Yaskawa INFORM job: OK_R2_O7,1(180,-90)OKKR_COMOUT.JBI

/JOB
//NAME OK_R2_O7,1(180,-90)OKKR_COMOUT
///FOLDERNAME X4
//POS
///NPOS 62,62,62,4,0,0
///TOOL 0
///POSTYPE PULSE
///PULSE
C00000=-125435,-77622,-99768,3556,84592,-1364
C00001=-127461,5107,-41648,6005,105402,-2311
C00002=-127602,-5081,-33811,5791,95110,-2850
C00003=-127461,-1910,-29167,5755,93871,-2860
C00004=-127461,-2146,-28156,5750,93132,-2895
C00005=-127461,-2037,-28638,5753,93482,-2879
C00006=-127360,629,-26422,5741,93484,-2844
C00007=-127461,-2008,-28767,5752,93576,-2874
C00008=-103998,1569,-25784,1957,92494,4742
C00009=-103998,1725,-26420,1958,92965,4749
C00010=-103998,1431,-25178,1956,92049,4737
C00011=-103998,1527,-25606,1957,92361,4742
C00012=-104229,4022,-23485,1997,92343,4666
C00013=-103998,1569,-25784,1957,92494,4742
C00014=-86679,-5363,-42434,-983,99074,10321
C00015=-62381,-14690,-36345,-9691,68856,-1615
C00016=-59861,14391,-7375,-13691,69257,-1127
C00017=-59861,14324,-5508,-13799,68107,-994
C00018=-59861,14327,-5726,-13788,68239,-1009
C00019=-59003,16580,-3664,-14156,68277,-700
C00020=-59755,14625,-6291,-13788,68745,-1031
C00021=-56899,7873,-12330,-14940,69480,-85
C00022=-55561,14142,-1887,-19350,68569,3889
C00023=-55984,15101,-1014,-19198,68428,3753
C00024=-55363,11408,-6012,-19288,69688,3774
C00025=-80499,-60483,-73568,-30648,97810,39569
C00026=-157567,-32017,-43550,-5241,58907,29882
C00027=-159996,-19727,-31763,-3894,57836,28984
C00028=-159996,-19632,-29676,-3947,56602,29029
C00029=-159996,-19645,-29901,-3941,56733,29024
C00030=-161459,-17871,-28596,-3080,56777,28442
C00031=-159996,-19645,-29901,-3941,56733,29024
C00032=-162143,-27333,-35707,-2694,56268,28184
C00033=-172681,-22690,-29875,17242,58260,14469
C00034=-172217,-21488,-29011,16987,58245,14658
C00035=-172321,-29251,-38222,16755,59878,14872
C00036=-170408,-23967,-31499,12392,55434,14706
C00037=-173810,-15316,-27557,19160,62810,14938
C00038=-170769,-6668,-20835,17665,62424,16063
C00039=-175825,-34683,-42059,20272,62319,14051
C00040=-166969,-54255,-34798,10244,21853,14480
C00041=-158903,-38412,-25890,-18291,26979,29827
C00042=-164397,-33556,-23512,2003,33361,24818
C00043=-170768,-56544,-33416,31030,22960,3886
C00044=-164207,-68143,-67141,2531,61479,16355
C00045=-79680,-75357,-72042,-32019,81856,-6685
C00046=-58622,-2742,-23483,-15327,69388,-15208
C00047=-58657,12974,-6767,-15536,67243,-14934
C00048=-62250,22223,1809,-14026,66090,-16116
C00049=-55419,-2669,-22327,-16741,69351,-14036
C00050=-47481,-9553,-15824,-35272,55767,14560
C00051=-66607,-8323,-12437,3279,42530,-8847
C00052=-66424,-8718,-12364,3138,42277,-8766
C00053=-66424,-7242,-5690,3358,38933,-8897
C00054=-61045,-16419,-29917,-8636,63731,-1843
C00055=-128613,-3227,-31039,5936,94424,-3210
C00056=-127935,508,-25861,5822,93118,-3048
C00057=-127978,405,-27754,5840,94227,-3010
C00058=-128179,-4770,-30252,5859,93124,-3128
C00059=-103810,3962,-22936,1928,91967,4796
C00060=-103028,-2446,-34673,1809,95878,5107
C00061=-101377,-7611,-58668,1615,107954,5791
BC00000=203857,716034,897320
BC00001=194529,717607,1053854
BC00002=194529,717607,1053854
BC00003=194529,717607,1053854
BC00004=194529,717607,1053854
BC00005=194529,717607,1053854
BC00006=194529,717607,1053854
BC00007=194529,717607,1053854
BC00008=194529,717607,1053854
BC00009=194529,717607,1053854
BC00010=194529,717607,1053854
BC00011=194529,717607,1053854
BC00012=194529,717607,1053854
BC00013=194529,717607,1053854
BC00014=194529,717607,1053854
BC00015=194529,709946,905441
BC00016=194529,709946,905441
BC00017=194529,709946,905441
BC00018=194529,709946,905441
BC00019=194529,709946,905441
BC00020=194529,709946,905441
BC00021=194529,709946,905441
BC00022=194529,709946,905441
BC00023=194529,709946,905441
BC00024=194529,709946,905441
BC00025=194529,709946,905441
BC00026=194529,709946,905441
BC00027=194529,709946,905441
BC00028=194529,709946,905441
BC00029=194529,709946,905441
BC00030=194529,709946,905441
BC00031=194529,709946,905441
BC00032=194529,709946,905441
BC00033=194529,709946,905441
BC00034=194529,709946,905441
BC00035=194529,709946,905441
BC00036=194529,709946,905441
BC00037=194529,709946,905441
BC00038=194529,709946,905441
BC00039=194529,709946,905441
BC00040=194529,709946,905441
BC00041=194529,709946,905437
BC00042=194529,709946,905437
BC00043=194529,709946,905441
BC00044=194529,709946,905441
BC00045=194529,709946,905441
BC00046=194529,709946,905441
BC00047=194529,709946,905441
BC00048=194529,709946,905441
BC00049=194529,709946,905441
BC00050=194529,709946,905441
BC00051=194529,709946,905441
BC00052=194529,709946,905441
BC00053=194529,709946,905441
BC00054=194529,709946,905441
BC00055=194529,717607,1053854
BC00056=194529,717607,1053854
BC00057=194529,717607,1053854
BC00058=194529,717607,1053854
BC00059=194529,717607,1053854
BC00060=194529,717607,1053854
BC00061=194529,717607,1053854
EC00000=1444023,-556474
EC00001=1319431,-556474
EC00002=1319431,-556474
EC00003=1319431,-556474
EC00004=1319431,-556474
EC00005=1319431,-556474
EC00006=1319431,-556474
EC00007=1319431,-556474
EC00008=1319431,-556474
EC00009=1319431,-556474
EC00010=1319431,-556474
EC00011=1319431,-556474
EC00012=1319431,-556474
EC00013=1319431,-556474
EC00014=1319431,-556474
EC00015=1506869,-556474
EC00016=1506869,-556474
EC00017=1506869,-556474
EC00018=1506869,-556474
EC00019=1506869,-556474
EC00020=1506869,-556474
EC00021=1506869,-556474
EC00022=1506869,-556474
EC00023=1506869,-556474
EC00024=1506869,-556474
EC00025=1506869,-556474
EC00026=1506869,-556474
EC00027=1506869,-556474
EC00028=1506869,-556474
EC00029=1506869,-556474
EC00030=1506869,-556474
EC00031=1506869,-556474
EC00032=1506869,-556474
EC00033=1506869,-556474
EC00034=1506869,-556474
EC00035=1506869,-556474
EC00036=1506869,-556474
EC00037=1506869,-556474
EC00038=1506869,-556474
EC00039=1506869,-556474
EC00040=1506869,-556474
EC00041=1506869,-556474
EC00042=1506869,-556474
EC00043=1506869,-556474
EC00044=1506869,-556474
EC00045=1506869,-556474
EC00046=1506869,-556474
EC00047=1506869,-556474
EC00048=1506869,-556474
EC00049=1506869,-556474
EC00050=1506869,-556474
EC00051=1506869,-556474
EC00052=1506869,-556474
EC00053=1506869,-556474
EC00054=1506869,-556474
EC00055=1319431,-556474
EC00056=1319431,-556474
EC00057=1319431,-556474
EC00058=1319431,-556474
EC00059=1319431,-556474
EC00060=1319431,-556474
EC00061=1319431,-556474
///POSTYPE BASE
///RECTAN
///RCONF 0,0,0,0,0,0,0,0,0,0,0,0,0,0,0,0,0,0,0,0,0,0,0,0
P00006=0.222,-3.123,-1.508,0.0000,0.0000,0.0000
P00021=-0.225,-6.128,-0.405,0.0000,0.0000,0.0000
P00040=-0.030,9.648,2.467,0.0000,0.0000,0.0000
P00041=0.192,3.924,0.305,0.0000,0.0000,0.0000
//INST
///DATE 2024/10/03 09:02
///ATTR SC,RW
///GROUP1 RB1,BS1
///GROUP2 ST1
NOP
'OK_r2_O7.1(180,-90)
'Path S1428
SFTOF3D
MOVJ C00000 BC00000 VJ=100.00  +MOVJ EC00000 VJ=100.00
MOVJ C00001 BC00001 VJ=100.00  +MOVJ EC00001 VJ=100.00
MOVJ C00002 BC00002 VJ=100.00  +MOVJ EC00002 VJ=100.00
SMOVL C00003 BC00003 V=100.0  +MOVJ EC00003
SREFP 3 C00004 BC00004  +REFP EC00004
CALL JOB:SEARCH-R1-S13D
SET P021 P006
SFTON3D P021
SMOVL C00005 BC00005 V=100.0  +MOVJ EC00005
SREFP 3 C00006 BC00006  +REFP EC00006
CALL JOB:SEARCH-R1-S13D
SET P021 P006
SFTON3D P021
SMOVL C00007 BC00007 V=100.0  +MOVJ EC00007
MOVL C00008 BC00008 V=1000.0  +MOVJ EC00008 VJ=100.00
SMOVL C00009 BC00009 V=100.0  +MOVJ EC00009
SREFP 3 C00010 BC00010  +REFP EC00010
CALL JOB:SEARCH-R1-S13D
SET P021 P006
SFTON3D P021
SMOVL C00011 BC00011 V=100.0  +MOVJ EC00011
SREFP 3 C00012 BC00012  +REFP EC00012
CALL JOB:SEARCH-R1-S13D
SET P021 P006
SFTON3D P021
SMOVL C00013 BC00013 V=100.0  +MOVJ EC00013
MOVJ C00014 BC00014 VJ=50.00  +MOVJ EC00014 VJ=50.00
MOVJ C00015 BC00015 VJ=50.00  +MOVJ EC00015 VJ=50.00
SFTOF3D
SMOVL C00016 BC00016 V=166.7  +MOVJ EC00016
SREFP 3 C00017 BC00017  +REFP EC00017
CALL JOB:SEARCH-R1-S13D
SET P040 P006
SFTON3D P040
SMOVL C00018 BC00018 V=100.0  +MOVJ EC00018
SREFP 3 C00019 BC00019  +REFP EC00019
CALL JOB:SEARCH-R1-S13D
SET P040 P006
SFTON3D P040
SMOVL C00020 BC00020 V=100.0  +MOVJ EC00020
SMOVL C00021 BC00021 V=166.7  +MOVJ EC00021
SMOVL C00022 BC00022 V=166.7  +MOVJ EC00022
SREFP 3 C00023 BC00023  +REFP EC00023
CALL JOB:SEARCH-R1-S13D
SET P040 P006
SFTON3D P040
SMOVL C00024 BC00024 V=166.7  +MOVJ EC00024
SFTOF3D
MOVJ C00025 BC00025 VJ=50.00  +MOVJ EC00025 VJ=50.00
MOVJ C00026 BC00026 VJ=50.00  +MOVJ EC00026 VJ=50.00
SMOVL C00027 BC00027 V=166.7  +MOVJ EC00027
SREFP 3 C00028 BC00028  +REFP EC00028
CALL JOB:SEARCH-R1-S13D
SET P041 P006
SFTON3D P041
SMOVL C00029 BC00029 V=100.0  +MOVJ EC00029
SREFP 3 C00030 BC00030  +REFP EC00030
CALL JOB:SEARCH-R1-S13D
SET P040 P041
SFTON3D P041
SMOVL C00031 BC00031 V=100.0  +MOVJ EC00031
SMOVL C00032 BC00032 V=166.7  +MOVJ EC00032
SMOVL C00033 BC00033 V=166.7  +MOVJ EC00033
SREFP 3 C00034 BC00034  +REFP EC00034
CALL JOB:SEARCH-R1-S13D
SET P041 P006
SFTON3D P041
SMOVL C00035 BC00035 V=166.7  +MOVJ EC00035
SFTOF3D
SFTON3D P041
MACRO1 MJ#(0) ARGF14
SMOVL C00036 BC00036 V=166.7  +MOVJ EC00036
ARCON
SMOVL C00037 BC00037 V=8.3  +MOVJ EC00037
SMOVL C00038 BC00038 V=8.3  +MOVJ EC00038
ARCOF
SMOVL C00039 BC00039 V=250.0  +MOVJ EC00039
SMOVL C00040 BC00040 V=250.0  +MOVJ EC00040
SMOVL C00041 BC00041 V=133.3 PL=0  +MOVJ EC00041
ARCON
SMOVL C00042 BC00042 V=9.2  +MOVJ EC00042
ARCOF
SMOVL C00043 BC00043 V=250.0  +MOVJ EC00043
MOVJ C00044 BC00044 VJ=50.00  +MOVJ EC00044 VJ=50.00
MOVJ C00045 BC00045 VJ=50.00  +MOVJ EC00045 VJ=50.00
MOVJ C00046 BC00046 VJ=50.00  +MOVJ EC00046 VJ=50.00
SFTON3D P040
SMOVL C00047 BC00047 V=166.7  +MOVJ EC00047
ARCON
SMOVL C00048 BC00048 V=8.3  +MOVJ EC00048
ARCOF
SMOVL C00049 BC00049 V=250.0  +MOVJ EC00049
SMOVL C00050 BC00050 V=250.0  +MOVJ EC00050
SMOVL C00051 BC00051 V=250.0  +MOVJ EC00051
ARCON
SMOVL C00052 BC00052 V=9.2  +MOVJ EC00052
SMOVL C00053 BC00053 V=9.2  +MOVJ EC00053
ARCOF
SMOVL C00054 BC00054 V=250.0  +MOVJ EC00054
MOVL C00055 BC00055 V=1000.0  +MOVJ EC00055 VJ=100.00
'Path W1429
'SPRAWDZ SZCZELNE
SFTOF3D
SFTON3D P021
SWVON WEV#(14)
SMOVL C00056 BC00056 V=100.0 PL=0  +MOVJ EC00056
SREFP 1 C00057 BC00057  +REFP EC00057
SREFP 2 C00058 BC00058  +REFP EC00058
MACRO1 MJ#(0) ARGF9
ARCON
SMOVL C00059 BC00059 V=8.3  +MOVJ EC00059
ARCOF
SWVOF
SMOVL C00060 BC00060 V=400.0  +MOVJ EC00060
SMOVL C00061 BC00061 V=1000.0  +MOVJ EC00061
SFTOF3D
END
